// TwinCAT 3 PLC project B5PIDController_Plc
// Title: B5PIDController_Plc
// Company: Tc3 Project
// ProjectVersion: 1.0.0.0
// ProgramVersion: 3.1.4026.22
// libraries:
//   Tc2_Standard, * (Beckhoff Automation GmbH)
//   Tc2_System, * (Beckhoff Automation GmbH)
// project tree:
//   / PlcTask.TcTTO
//   POUs/ FB_PIDController.TcPOU, MAIN.TcPOU
// real-time tasks:
//   TASK PlcTask: cycle T#10ms, priority 20, ADS port 350

CONFIGURATION B5PIDController_Plc
    RESOURCE PLC ON TwinCAT3
        TASK PlcTask(INTERVAL := T#10ms, PRIORITY := 20);
        PROGRAM MAIN WITH PlcTask : MAIN;
    END_RESOURCE
END_CONFIGURATION

// ---- POUs/MAIN.TcPOU
PROGRAM MAIN
VAR
END_VAR

END_PROGRAM

// ---- POUs/FB_PIDController.TcPOU
FUNCTION_BLOCK FB_PIDController
VAR_INPUT
    fError : REAL;
END_VAR
VAR_OUTPUT
    fOutput : REAL;
END_VAR
VAR
    fGain : REAL := 0.0;
END_VAR

METHOD Step : REAL
VAR
END_VAR
fOutput := fError * fGain;
Step := fOutput;
END_METHOD

END_FUNCTION_BLOCK
